{attribute 'GeneratedUsingTerminal: EL5101--0000'}
{attribute addProperty BoxType "EL5101--0000"}
{attribute addProperty Id "StatusAT %I*USINT1ValueAT %I*UINT2LatchAT %I*UINT2"}
{attribute addProperty CRC "3104192441"}
{attribute addProperty Size "5"}
TYPE Channel_B90637B9 :
STRUCT
	{attribute addProperty Name "Status"}
	Status AT %I* : USINT;
	{attribute addProperty Name "Value"}
	Value AT %I* : UINT;
	{attribute addProperty Name "Latch"}
	Latch AT %I* : UINT;
END_STRUCT
END_TYPE

(* stored: Version 1.2.0.0, ProductVersion 3.1.4024.9
   DUT Channel_B90637B9: Id {3676019c-0198-44c8-b974-07df9629eeb4} *)
